TYPE TcoDiConfig :
STRUCT
	IsFalseTimeOut : TIME := T#10S;
	IsTrueTimeOut : TIME := T#10S;
END_STRUCT
END_TYPE

(* stored: Version 1.1.0.1, ProductVersion 3.1.4026.8
   DUT TcoDiConfig: Id {94f7ac71-8bb7-00e4-3f17-566f5e98c292} *)
